// TwinCAT 3 PLC project main
// ProgramVersion: 3.1.4023.0
// libraries:
//   Tc2_Standard, * (Beckhoff Automation GmbH)
//   Tc3_Module, * (Beckhoff Automation GmbH)
//   Tc2_System,3.4.21.0,Beckhoff Automation GmbH
// project tree:
//   DUTs/ E_DataSet.TcDUT, ST_DataPoint.TcDUT, E_ProgramState.TcDUT
//   GVLs/ GVL.TcGVL
//   / PlcTask.TcTTO
//   POUs/ MAIN.TcPOU
// real-time tasks:
//   TASK PlcTask: cycle T#1ms, priority 20, ADS port 350

CONFIGURATION main
    RESOURCE PLC ON TwinCAT3
        TASK PlcTask(INTERVAL := T#1ms, PRIORITY := 20);
        PROGRAM MAIN WITH PlcTask : MAIN;
    END_RESOURCE
END_CONFIGURATION

// ---- DUTs/E_DataSet.TcDUT
{attribute 'qualified_only'}
{attribute 'strict'}
TYPE E_DataSet :
(
	SETPOINTS := 1,
	ACTUAL := 2
);
END_TYPE

// ---- DUTs/ST_DataPoint.TcDUT
TYPE ST_DataPoint :
STRUCT

	x : INT;
	y : INT;

END_STRUCT
END_TYPE

// ---- DUTs/E_ProgramState.TcDUT
{attribute 'qualified_only'}
{attribute 'strict'}
TYPE E_ProgramState :
(
	INIT,
	REFRESH_SETPOINTS_USING_FORMULA,
	WAIT_FOR_START_COMMAND,
	ACTIVE,
	COMPLETE,
	RESET	
);
END_TYPE

// ---- GVLs/GVL.TcGVL
VAR_GLOBAL CONSTANT

	MAX_POINTS : INT := 600;	

END_VAR
VAR_GLOBAL

	programState : E_ProgramState := E_ProgramState.INIT;
	dataPoints : ARRAY[1..2, 0..MAX_POINTS] OF ST_DataPoint;

END_VAR

// ---- POUs/MAIN.TcPOU
PROGRAM MAIN
VAR
	
	i : INT; 
	
	// used to create the bell curve
	a : LREAL := 200;
	b : LREAL := 4;
	c : LREAL := 300;
	
	yScale : LREAL := 700;
	
	delayTimer : ton;
	activePoint : INT;
	tempSetpoint : INT;
	randomNumberGenerator : DRAND;
	randomNumber : LREAL;
	
END_VAR

CASE GVL.programState OF
	
	E_ProgramState.INIT:
	
		// quick method of cleaning an array
		memset(ADR(GVL.dataPoints),16#0,SIZEOF(GVL.dataPoints));
		activePoint := 0;
		
		// move to next state
		GVL.programState := E_ProgramState.REFRESH_SETPOINTS_USING_FORMULA;
	
	E_ProgramState.REFRESH_SETPOINTS_USING_FORMULA:
		
		// setup a bell curve in the setpoint datapoint array
		FOR i := 0 TO GVL.MAX_POINTS DO
			
			GVL.dataPoints[E_DataSet.SETPOINTS,i].x := i;
			GVL.dataPoints[E_DataSet.SETPOINTS,i].y := LREAL_TO_INT((1 / (1 + (EXPT(((GVL.dataPoints[E_DataSet.SETPOINTS,i].x-c)/a),(2 * b))))) * yScale);
		
		END_FOR
		
		// move to next state
		GVL.programState := E_ProgramState.WAIT_FOR_START_COMMAND;
	
	E_ProgramState.WAIT_FOR_START_COMMAND:
	
		// the hmi will trigger the program state to change to active when the start button is pressed.
	
	E_ProgramState.ACTIVE:
	
		delayTimer(pt:=T#100MS, in:=NOT delayTimer.Q);
		

		IF delayTimer.Q THEN
			IF activePoint <= GVL.MAX_POINTS THEN 
				activePoint := activePoint + 1;
				
				// read an actual value an place in the array.
				// for this example the actual value is the setpoint + some random noise
				
				tempSetpoint := GVL.dataPoints[E_DataSet.SETPOINTS,activePoint].y;
				randomNumber := randomNumberGenerator.Num;
				tempSetpoint := tempSetpoint - LREAL_TO_INT((randomNumber*20)-10);
				
				GVL.dataPoints[E_DataSet.ACTUAL,activePoint].x := activePoint;
				GVL.dataPoints[E_DataSet.ACTUAL,activePoint].y := tempSetpoint;
				
				FOR i := activePoint TO GVL.MAX_POINTS DO
					GVL.dataPoints[E_DataSet.ACTUAL,i].x := activePoint;
					GVL.dataPoints[E_DataSet.ACTUAL,i].y := tempSetpoint;
				END_FOR
				
				
			ELSE
				GVL.programState := E_ProgramState.COMPLETE;
			END_IF
			
		END_IF
	
	E_ProgramState.COMPLETE:
	
	E_ProgramState.RESET:
	
		// user selects reset so re-init
		GVL.programState := E_ProgramState.INIT;
	
END_CASE

randomNumberGenerator(seed:=0);

END_PROGRAM
